/// Implicitly generated code : DO NOT EDIT!!!
/// Checks for division by 0, if divisor is 0, replace it with 1 and report error
{attribute 'no_check' := ''}
{attribute 'check_div_int64' := ''}
FUNCTION CheckDivLInt : LINT
VAR_INPUT
	divisor: LINT;
END_VAR

IF divisor = 0 THEN
	// replace divisor and report error if necessary
	CheckDivLInt := 1;
	GVL_Supervision.aCodeErr[eCodeError_divLInt] := TRUE;
ELSE
	CheckDivLInt := divisor;
END_IF;

END_FUNCTION

(* stored: Version 1.1.0.1, ProductVersion 3.1.4022.9
   POU CheckDivLInt: Id {a0ba4f07-7587-44a7-aef9-ee47a1cc821d}, SpecialFunc None *)
